Staubli VAL3: stop.pgx

program stop()
begin
  //当程序运行完会自动调用stop程序
  //当按下stop键时会调用stop程序
  popUpMsg("调用stop程序")


end
